(* IEC 61131-3 sources: programs/VI-54/VI-54_20171205/VI-54_20171205/Stations/Screen/LseClass170718/Class/HourCounter, 1 file *)

(* ---- HourCounter.st ---- *)
(*!
<Class
	Name               = "HourCounter"
	Revision           = "0.0"
	RealtimeTask       = "false"
	CyclicTask         = "false"
	BackgroundTask     = "true"
	Sigmatek           = "false"
	OSInterface        = "false"
	HighPriority       = "false"
	Automatic          = "false"
	UpdateMode         = "Prescan"
	SharedCommandTable = "true"
	Objectsize         = "(840,120)">
	<Channels>
		<Server Name="ClassSvr" Visualized="false" Initialize="false" WriteProtected="true" Retentive="false"/>
		<Server Name="GraphActive" Visualized="true" Initialize="true" WriteProtected="false" Retentive="File"/>
		<Server Name="ResetData" Visualized="true" Initialize="false" WriteProtected="false" Retentive="false"/>
		<Client Name="iClock" Required="true" Internal="false"/>
		<Client Name="Standard6" Required="true" Internal="true"/>
	</Channels>
	<Network Name="HourCounter">
		<!-- List of Components in this network -->
		<Components>
			<Object
				Name           = "Standard6"
				Class          = "Standard"
				Position       = "(270,390)"
				Visualized     = "false"
				BackgroundTime = "1000 ms">
				<Channels>
					<Server Name="ClassSvr"/>
				</Channels>
			</Object>
		</Components>
		<Comments>
		</Comments>
		<!-- List of Connections in this network -->
		<Connections>
			<Connection Source="this.Standard6" Destination="Standard6.ClassSvr"/>
		</Connections>
		<!-- Headerfiles -->
		<Options>
		</Options>
	</Network>
</Class>
*)
HourCounter : CLASS
  //Servers:
	ClassSvr 	: SvrChCmd_DINT;
	ResetData 	: SvrCh_DINT;
	GraphActive 	: SvrCh_OptiesEnum;
  //Clients:
	iClock 	: CltChCmd_DateAndTime;
	Standard6 	: CltChCmd_Standard;
  //Variables:
		HourStr 	: HourCntrStr;
		NbrOfPackets 	: DINT;
		MinutsOfRunning 	: DINT;
		OldMinute 	: DINT;
		OldHour 	: DINT;
		ActRunStatus 	: RunningStateEnum;
		ActNbrOfPackets 	: DINT;
		ResetCntrs 	: DINT;
  //Functions:

	FUNCTION VIRTUAL GLOBAL Background
		VAR_INPUT
			EAX 	: UDINT;
		END_VAR
		VAR_OUTPUT
			state (EAX) 	: UDINT;
		END_VAR;

	FUNCTION GLOBAL GetValue
		VAR_OUTPUT
			Data 	: HourCntrStr;
		END_VAR;

	FUNCTION GLOBAL GetRunState
		VAR_INPUT
			RunState 	: RunningStateEnum;
		END_VAR;

	FUNCTION GLOBAL GetPacketCntr
		VAR_INPUT
			Cntr 	: DINT;
		END_VAR;

	FUNCTION GLOBAL ResetCounters
		VAR_INPUT
			ReadReset 	: DINT;
		END_VAR
		VAR_OUTPUT
			Reset 	: DINT;
		END_VAR;
  //Tables:
	FUNCTION @STD
		VAR_OUTPUT
			ret_code	: CONFSTATES;
		END_VAR;
	FUNCTION GLOBAL TAB @CT_;
END_CLASS;

#pragma using Standard
#pragma usingLtd DateAndTime

FUNCTION VIRTUAL GLOBAL HourCounter::Background
	VAR_INPUT
		EAX 	: UDINT;
	END_VAR
	VAR_OUTPUT
		state (EAX) 	: UDINT;
	END_VAR
  VAR
  	xxx : Dint;
  END_VAR

  // Reset the data
  if ResetData = 1 then
    for xxx := 0 to ((sizeof(HourCntrStr) / sizeof(CntrStr)) - 1) do
      HourStr[xxx].MinutsOfRunning := 0;
      HourStr[xxx].NbrOfPackets := 0;
    end_for;
    ResetCntrs := 1;
    ResetData := 0;
  end_if;

  if ActNbrOfPackets <> NbrOfPackets then
    NbrOfPackets := ActNbrOfPackets;
  end_if;

  if ActRunStatus = eRunStatus then
    if OldMinute <> iClock.Minute then
      MinutsOfRunning += 1;
      OldMinute := iClock.Minute;
    end_if;
  end_if;

  if iClock.Hour <> OldHour then
    HourStr[iClock.Hour].MinutsOfRunning := MinutsOfRunning;
    HourStr[iClock.Hour].NbrOfPackets := NbrOfPackets;
    // reset the counters
    ResetCntrs := 1;
    MinutsOfRunning := 0;
    NbrOfPackets := 0;
    OldHour := iClock.Hour;
  end_if;

	state := READY;

END_FUNCTION

FUNCTION GLOBAL HourCounter::GetValue
	VAR_OUTPUT
		Data 	: HourCntrStr;
	END_VAR

  Data := HourStr;

END_FUNCTION

FUNCTION GLOBAL HourCounter::GetRunState
	VAR_INPUT
		RunState 	: RunningStateEnum;
	END_VAR

  ActRunStatus := RunState;

END_FUNCTION

FUNCTION GLOBAL HourCounter::GetPacketCntr
	VAR_INPUT
		Cntr 	: DINT;
	END_VAR

  ActNbrOfPackets := Cntr;

END_FUNCTION

FUNCTION GLOBAL HourCounter::ResetCounters
	VAR_INPUT
		ReadReset 	: DINT;
	END_VAR
	VAR_OUTPUT
		Reset 	: DINT;
	END_VAR

  // Reset counters
  if ReadReset = 1 then
    ResetCntrs := 0;
  else
    Reset := ResetCntrs;
  end_if;

END_FUNCTION
